PROGRAM Scaling
VAR
END_VAR
// written 10.07.2023 by Daniel Kelly

// Program provides scaling for the signals from the thermocouples

drive.ScaledThermoCouple1Value := drive.RawThermoCouple1Value * (1000.0/32767); // not in use
drive.ScaledThermoCouple2Value := drive.RawThermoCouple2Value * (1000.0/32767);

END_PROGRAM

(* stored: Version 1.1.0.1, ProductVersion 3.1.4024.12
   POU Scaling: Id {49c2dd34-2ec2-4425-9c62-41867a3fdf38}, SpecialFunc None *)
